(* CoDeSys 2.3 export: SIRENA.EXP *)

(* POU sirenStart, CFC *)
PROGRAM sirenStart
VAR
	tpStart: TP;
	blnk: BLINK;
	zvon: BOOL;
	trig: F_TRIG;
END_VAR
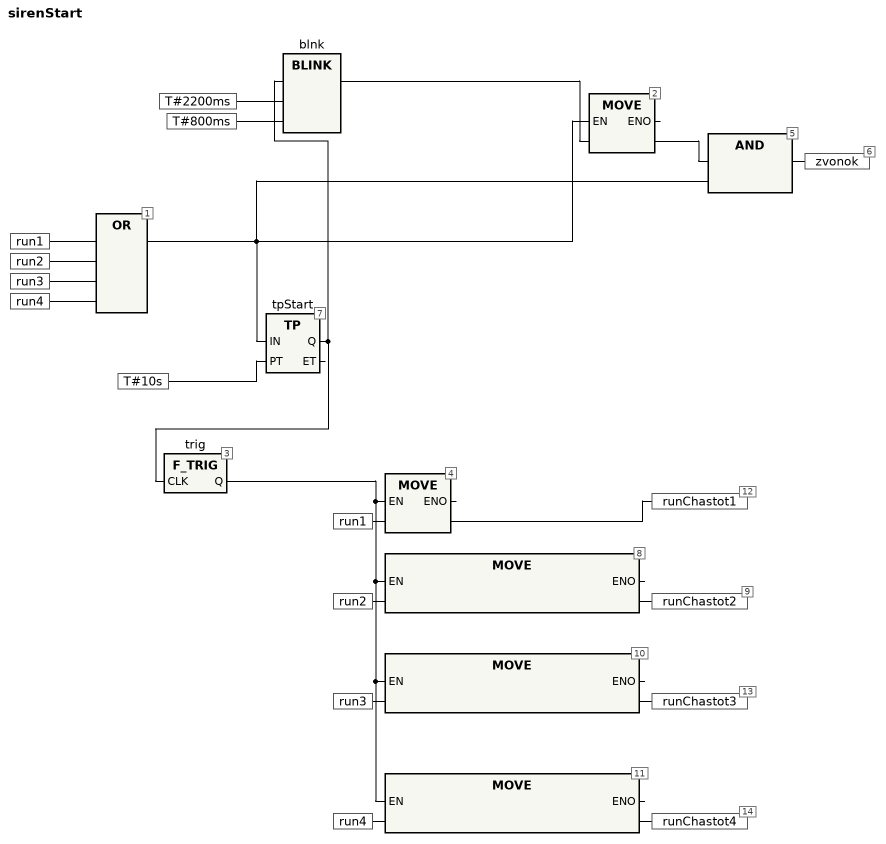
_CFC_ (* Continuous Function Chart, elements in execution order *)
#0 blnk:BLINK(#7.Q, T#2200ms, T#800ms)
#1 OR(run1, run2, run3, run4)
#2 MOVE(EN: #1, #0)
#3 trig:F_TRIG(CLK: #7.Q)
#4 MOVE(EN: #3.Q, run1)
#5 AND(#2, #1)
#6 zvonok <= #5
#7 tpStart:TP(IN: #1, PT: T#10s)
#8 MOVE(EN: #3.Q, run2)
#9 runChastot2 <= #8
#10 MOVE(EN: #3.Q, run3)
#11 MOVE(EN: #3.Q, run4)
#12 runChastot1 <= #4
#13 runChastot3 <= #10
#14 runChastot4 <= #11
_END_CFC_
END_PROGRAM

(* POU sirenStop, CFC *)
PROGRAM sirenStop
VAR
	tpStop: TP;
	zvon: BOOL;
	trig: R_TRIG;
	firstTime: BOOL;
END_VAR
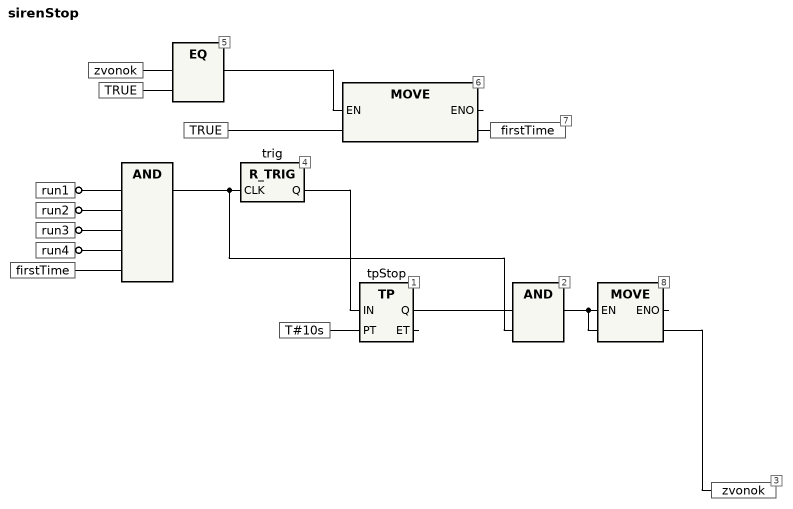
_CFC_ (* Continuous Function Chart, elements in execution order *)
#0 AND(NOT run1, NOT run2, NOT run3, NOT run4, firstTime)
#1 tpStop:TP(IN: #4.Q, PT: T#10s)
#2 AND(#1.Q, #0)
#3 zvonok <= #8
#4 trig:R_TRIG(CLK: #0)
#5 EQ(zvonok, TRUE)
#6 MOVE(EN: #5, TRUE)
#7 firstTime <= #6
#8 MOVE(EN: #2, #2)
_END_CFC_
END_PROGRAM
